FUNCTION_BLOCK COURIER_CAT (* Composite Function Block Type *)
  (* Standard: 61499-2 *)
  (* Version 0.0, 12/17/2022, Dmitrii, Flexbridge AB, template *)
  PACKAGE Main;
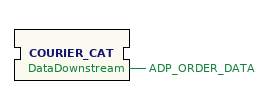
  PLUGS
    DataDownstream : ADP_ORDER_DATA;
  END_PLUGS
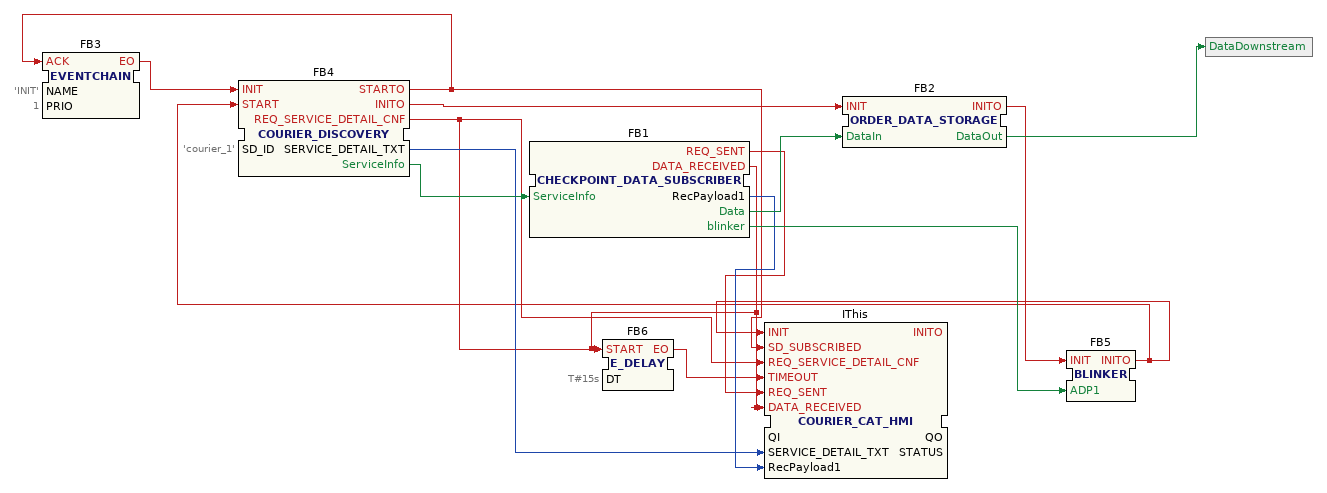
  (* HMI *)
  FBS
    FB1 : CHECKPOINT_DATA_SUBSCRIBER;
    FB2 : ORDER_DATA_STORAGE;
    FB4 : COURIER_DISCOVERY(SD_ID := 'courier_1');
    FB3 : EVENTCHAIN(NAME := 'INIT', PRIO := 1);
    FB5 : BLINKER;
    IThis : COURIER_CAT_HMI;
    FB6 : E_DELAY(DT := T#15s);
  END_FBS
  EVENT_CONNECTIONS
    FB3.EO TO FB4.INIT;
    FB4.STARTO TO FB3.ACK;
    FB4.INITO TO FB2.INIT;
    FB2.INITO TO FB5.INIT;
    FB5.INITO TO FB4.START;
    FB4.REQ_SERVICE_DETAIL_CNF TO FB6.START;
    FB5.INITO TO IThis.INIT;
    FB4.STARTO TO IThis.SD_SUBSCRIBED;
    FB4.REQ_SERVICE_DETAIL_CNF TO IThis.REQ_SERVICE_DETAIL_CNF;
    FB6.EO TO IThis.TIMEOUT;
    FB1.REQ_SENT TO IThis.REQ_SENT;
    FB1.DATA_RECEIVED TO IThis.DATA_RECEIVED;
    FB1.DATA_RECEIVED TO FB6.START;
  END_CONNECTIONS
  DATA_CONNECTIONS
    FB4.SERVICE_DETAIL_TXT TO IThis.SERVICE_DETAIL_TXT;
    FB1.RecPayload1 TO IThis.RecPayload1;
  END_CONNECTIONS
  ADAPTER_CONNECTIONS
    FB1.Data TO FB2.DataIn;
    FB1.blinker TO FB5.ADP1;
    FB2.DataOut TO DataDownstream;
    FB4.ServiceInfo TO FB1.ServiceInfo;
  END_CONNECTIONS
END_FUNCTION_BLOCK
